FUNCTION FILE_PATH_SPLIT : BOOL
VAR_INPUT
	FILENAME : T_MaxString;
END_VAR
VAR_IN_OUT
	X : FILE_PATH_DATA;
END_VAR
VAR
	b : INT;
	c : INT;
	d : STRING(1);
	p1 : INT;
	p2 : INT;
END_VAR

(*
version 1.0		01. jan. 2011
programmer		ks
tested by			ks

FILE_PATH_SPLIT zerlegt einen Dateipfad in einzelne Elemente und legt diese in einer Datenstruktur ab.
*)

X.DRIVE := '';
X.DIRECTORY := '';
X.FILENAME := '';
c := LEN(FILENAME);
IF c = 0 THEN
	FILE_PATH_SPLIT := FALSE;
	RETURN;
END_IF;

FOR b := 1 TO c DO
	d := MID(FILENAME, 1, b);
	IF d = ':' THEN
		p1 := b;
	ELSIF d = '/' OR d = '\' THEN
		p2 := b;
	END_IF;
END_FOR;

IF p1 = 2 THEN
	X.DRIVE := LEFT(FILENAME,p1);
END_IF;

IF p2 > 0 AND p2 > p1 THEN
	X.DIRECTORY := MID(FILENAME,p2 - p1,p1+1); (* len , pos *)
END_IF;

X.FILENAME := RIGHT(FILENAME,c - MAX (p1,p2));
FILE_PATH_SPLIT := TRUE;

(* revision history
ks	01. jan. 2011	rev 1.0
	original version
*)

END_FUNCTION

(* stored: Version 1.1.0.1, ProductVersion 3.1.4024.9
   POU FILE_PATH_SPLIT: Id {0dee58bc-420b-4208-b2c5-7330a48045eb}, SpecialFunc None *)
